// TIA Portal V16 export
// export: Created 2023-03-29T11:03:41.9730188Z, ExportSetting WithDefaults, DisplayName Totally Integrated Automation Portal, DisplayVersion V16 Update 6, DisplayName TIA Portal Version Control Interface, DisplayVersion V16 Update 2, DisplayName TIA Portal Openness, DisplayVersion V16 Update 6, DisplayName STEP 7 Professional, DisplayVersion V16 Update 6, DisplayName STEP 7 Safety, DisplayVersion V16, DisplayName WinCC Advanced, DisplayVersion V16 Update 6
DATA_BLOCK "generator_weekday_DB"   // DB49
AUTHOR : RTecmer
FAMILY : XMHour
VERSION : 0.1
// stored: AutoNumber true, DBAccessibleFromOPCUA true, InstanceOfName generator_weekday, InstanceOfType FB
"generator_weekday"
   // VAR_INPUT
   //    Reset { ExternalAccessible := 'False'; ExternalVisible := 'False'; ExternalWritable := 'False'} : Bool;
   //    Run_WEEKDAY : Bool;
   // END_VAR
   // VAR_OUTPUT
   //    Out_Weekday : Bool;
   // END_VAR
   // VAR_IN_OUT
   //    Data_sek : Int;
   //    Data_hour : DWord;
   //    Edge_Hz { ExternalAccessible := 'False'; ExternalVisible := 'False'; ExternalWritable := 'False'} : Bool;
   // END_VAR
   // VAR
   //    sek_real { ExternalAccessible := 'False'; ExternalVisible := 'False'; ExternalWritable := 'False'} : Real;
   //    hour_sek { ExternalAccessible := 'False'; ExternalVisible := 'False'; ExternalWritable := 'False'} : Real;
   //    memTrig_Week : Bool;
   //    start_weekday : Bool;
   //    tmp_weekend : USInt;
   // END_VAR
BEGIN
END_DATA_BLOCK
